FUNCTION_BLOCK FB_Server
VAR_OUTPUT
	bValid : BOOL;
END_VAR
VAR
	_fbServer 	: FB_OCPP1_Server(0);
	// receive
	hStationId 	: UDINT;
	hMessageId 	: T_OCPP_MessageId;
	eAction 	: E_OCPP1_Action;
END_VAR

METHOD Execute : BOOL
bValid := _fbServer.bValid;
IF NOT bValid THEN RETURN; END_IF
END_METHOD

METHOD FB_Init : BOOL
VAR_INPUT
	bInitRetains : BOOL; // if TRUE, the retain variables are initialized (warm start / cold start)
	bInCopyCode : BOOL;  // if TRUE, the instance afterwards gets moved into the copy code (online change)

	stParam : REFERENCE TO ST_OCPP1_ServerParam;
END_VAR
IF bInCopyCode THEN RETURN; END_IF

FB_Init := _fbServer.Init(stParam);
END_METHOD

PROPERTY Server : REFERENCE TO FB_OCPP1_Server
GET
Server REF= _fbServer;
END_GET
END_PROPERTY

END_FUNCTION_BLOCK

(* stored: Version 1.1.0.1
   POU FB_Server: Id {1bf0250d-b6d0-4041-bd86-279312d44979}, SpecialFunc None
   Method Execute: Id {f894dc41-ef8a-47cb-8749-d4fe3d89ca14}
   Method FB_Init: Id {9659b0af-8b27-4926-8c1b-4473f332beef}
   Property Server: Id {759de8ec-c984-4874-8b4d-a9783312f1ca}
   Get Get: Id {77c772a7-e96f-4fae-be82-0f1b286a197d} *)
